// TIA Portal project "DrillingMachineS7300_S71500" (V15.1)

(* hardware
DEVICE "S7300/ET200M-Station_1"  S7-300 station
   slot 0: "Profilschiene_0"  Rail  6ES7 390-1***0-0AA0
   slot 2: "PLC_1"  CPU 315-2 PN/DP  6ES7 315-2EH14-0AB0  V3.2
      slot 2: "PROFINET-Schnittstelle_1"  PN-IO
         slot 1: "Port_1"  Port
         slot 2: "Port_2"  Port
   slot 4: "DI 32x24VDC_1"  DI32 x 24VDC  6ES7 321-1BL00-0AA0
   slot 5: "DO 32x24VDC/0.5A_1"  DO32 x 24VDC / 0.5A  6ES7 322-1BL00-0AA0
   slot 6: "AI 2x12BIT_1"  AI2 x 12 bits  6ES7 331-7KB02-0AB0
   slot 7: "AO 4x12BIT_1"  AO4 x 12 bits  6ES7 332-5HD01-0AB0
DEVICE "S71500/ET200MP-Station_1"  S7-1500 station
   slot 0: "Profilschiene_0"  Rack  6ES7 590-1***0-0AA0
   slot 1: "PLC_2"  CPU 1513-1 PN  6ES7 513-1AL02-0AB0  V2.6
      slot 3: "CPU-Display_1"  6ES7591-1AA00-0AA0
   slot 2: "DI 32x24VDC BA_1"  DI 32x24VDC BA  6ES7 521-1BL10-0AA0  V1.0
   slot 3: "DQ 32x24VDC/0.5A ST_1"  DQ 32x24VDC/0.5A ST  6ES7 522-1BL00-0AB0  V2.0
   slot 4: "AI 4xU/I/RTD/TC ST_1"  AI 4xU/I/RTD/TC ST  6ES7 531-7QD00-0AB0  V1.0
   slot 5: "AQ 4xU/I ST_1"  AQ 4xU/I ST  6ES7 532-5HD00-0AB0  V2.2
   slot 6: "DI 16x24VDC BA_1"  DI 16x24VDC BA  6ES7 521-1BH10-0AA0  V1.0
*)

// ===== PLC "PLC_1"  CPU 315-2 PN/DP =====

VAR_GLOBAL   // PLC tag table "Standard-Variablentabelle"
   "ControlOn" AT %M0.0 : Bool;
   "InitialPos" AT %M0.1 : Bool;
   "B14ClampingJaw1Min" AT %E2.6 : Bool;   // NC
   "B15ClampingJaw2Min" AT %E2.7 : Bool;   // NC
   "B16ClampingJaw3Min" AT %E3.0 : Bool;   // NC
   "B17ClampingJaw4Min" AT %E3.1 : Bool;   // NC
   "M13ClampingJawsToMax" AT %A2.5 : Bool;
END_VAR

VAR_GLOBAL   // PLC tag table "Variablentabelle aus XML_1"
   "S1ControlOn" AT %I0.0 : Bool;
   "S2ControlOff" AT %I0.1 : Bool;
   "S3Start" AT %I0.2 : Bool;
   "B1DrillMachVertMin" AT %I1.0 : Bool;   // NC
   "B2DrillMachVertMax" AT %I1.1 : Bool;   // NC
   "P1ControlOn" AT %Q0.0 : Bool;
   "M1DrillMachToMax" AT %Q1.0 : Bool;
   "M2DrillMachToMin" AT %Q1.1 : Bool;
   "M3DrillMachOn" AT %Q1.2 : Bool;
   "M4RotateDrillMachine" AT %Q1.3 : Bool;
   "RotationDrillMachStart" AT %Q1.4 : Bool;
   "B4DrillMachHorizMin" AT %I1.3 : Bool;   // NC
   "B3RotationDrillMachPos" AT %IW10 : Int;
   "RotationDrillMachNewPosReached" AT %I1.2 : Bool;
   "RotationDrillMachNewPos" AT %QW10 : Int;
   "B5DrillMachHorizMax" AT %I1.4 : Bool;   // NC
   "M5DrillMachHoriz" AT %Q1.5 : Bool;
   "DrillMachHorizStart" AT %Q1.6 : Bool;
   "B6FeedMinPos" AT %I1.5 : Bool;   // NC
   "B7FeedMaxPos" AT %I1.6 : Bool;   // NC
   "B8FeedDrillPos" AT %I1.7 : Bool;
   "M7FeedToMax" AT %Q1.7 : Bool;
   "M8FeedToMin" AT %Q2.0 : Bool;
   "M9GuideToMax" AT %Q2.1 : Bool;
   "M10GuideToMin" AT %Q2.2 : Bool;
   "B9GuideMinPos" AT %I2.0 : Bool;   // NC
   "B10GuideMaxPos" AT %I2.1 : Bool;   // NC
   "M11SliderToMax" AT %Q2.3 : Bool;
   "M12SliderToMin" AT %Q2.4 : Bool;
   "B11SliderMinPos" AT %I2.2 : Bool;   // NC
   "B12SliderMaxPos" AT %I2.3 : Bool;   // NC
   "B13MetalRodInSliderPos" AT %I2.4 : Bool;
   "B18DrillMachHorizPos" AT %IW12 : Word;
   "DrillMachHorizNewPos" AT %QW12 : Word;
   "DrillMachHorizNewPosReached" AT %I2.5 : Bool;
END_VAR

DATA_BLOCK "DrillMachineHorizPositioning_DB_FirstPos"   // DB1
{ S7_Optimized_Access := 'FALSE' }
VERSION : 0.1
// stored: InstanceOfName DrillMachineHorizPositioning
"DrillMachineHorizPositioning"
BEGIN
END_DATA_BLOCK

DATA_BLOCK "DrillMachineRotPositioning_DB_FirstPos"   // DB2
{ S7_Optimized_Access := 'FALSE' }
VERSION : 0.1
// stored: InstanceOfName DrillMachineRotationPositioning
"DrillMachineRotationPositioning"
BEGIN
END_DATA_BLOCK

DATA_BLOCK "DrillMachineHorizPositioning_DB_SecondPos"   // DB3
{ S7_Optimized_Access := 'FALSE' }
VERSION : 0.1
// stored: InstanceOfName DrillMachineHorizPositioning
"DrillMachineHorizPositioning"
BEGIN
END_DATA_BLOCK

DATA_BLOCK "DrillMachineRotPositioning_DB_SecondPos"   // DB4
{ S7_Optimized_Access := 'FALSE' }
VERSION : 0.1
// stored: InstanceOfName DrillMachineRotationPositioning
"DrillMachineRotationPositioning"
BEGIN
END_DATA_BLOCK

DATA_BLOCK "DrillMachineHorizPositioning_DB_ThirdPos"   // DB5
{ S7_Optimized_Access := 'FALSE' }
VERSION : 0.1
// stored: InstanceOfName DrillMachineHorizPositioning
"DrillMachineHorizPositioning"
BEGIN
END_DATA_BLOCK

DATA_BLOCK "DrillMachineRotPositioning_DB_ThirdPos"   // DB6
{ S7_Optimized_Access := 'FALSE' }
VERSION : 0.1
// stored: InstanceOfName DrillMachineRotationPositioning
"DrillMachineRotationPositioning"
BEGIN
END_DATA_BLOCK

DATA_BLOCK "StepsDB"   // DB7
{ S7_Optimized_Access := 'FALSE' }
VERSION : 0.1
// stored: InstanceOfName Steps
"Steps"
BEGIN
END_DATA_BLOCK

FUNCTION_BLOCK "Steps"   // FB1, FBD
{ S7_Optimized_Access := 'FALSE' }
VERSION : 0.1
   VAR
      NewPosHorizReachedHelper_0 : Bool;
      NewPosVertReachedHelper_0 : Bool;
      NewPosHorizReachedHelper_1 : Bool;
      NewPosVertReachedHelper_1 : Bool;
      NewPosHorizReachedHelper_2 : Bool;
      NewPosVertReachedHelper_2 : Bool;
      NewPosHorizReachedHelper_3 : Bool;
      NewPosVertReachedHelper_3 : Bool;
      Step1 : Bool;
      Step2 : Bool;
      Step3 : Bool;
      Step4 : Bool;
      Step5 : Bool;
      Step6 : Bool;
      Step7 : Bool;
      Step8 : Bool;
      Step9 : Bool;
      Step10 : Bool;
      Step11 : Bool;
      Step12 : Bool;
      Step12A : Bool;
      Step13 : Bool;
      Step14 : Bool;
      Step15 : Bool;
      Step15A : Bool;
      Step16 : Bool;
      Step17 : Bool;
      Step18 : Bool;
      Step19 : Bool;
      Step20 : Bool;
      InStepChain : Bool;
   END_VAR
   VAR_TEMP   // added for the SCL form of the ladder/FBD networks
      _w1 : Bool;
   END_VAR
BEGIN

REGION Network 1: Start
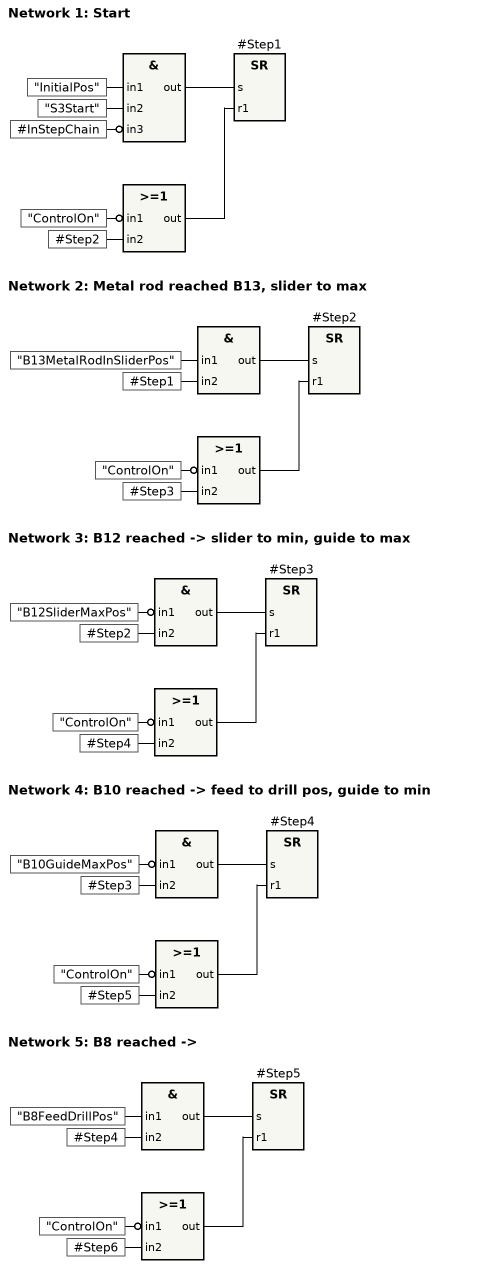
   IF "InitialPos" AND "S3Start" AND NOT #InStepChain THEN
       #Step1 := TRUE;   // SR flip-flop
   END_IF;
   IF NOT "ControlOn" OR #Step2 THEN #Step1 := FALSE; END_IF;
END_REGION

REGION Network 2: Metal rod reached B13, slider to max
   IF "B13MetalRodInSliderPos" AND #Step1 THEN
       #Step2 := TRUE;   // SR flip-flop
   END_IF;
   IF NOT "ControlOn" OR #Step3 THEN #Step2 := FALSE; END_IF;
END_REGION

REGION Network 3: B12 reached -> slider to min, guide to max
   // Slider stops with B11
   IF NOT "B12SliderMaxPos" AND #Step2 THEN
       #Step3 := TRUE;   // SR flip-flop
   END_IF;
   IF NOT "ControlOn" OR #Step4 THEN #Step3 := FALSE; END_IF;
END_REGION

REGION Network 4: B10 reached -> feed to drill pos, guide to min
   IF NOT "B10GuideMaxPos" AND #Step3 THEN
       #Step4 := TRUE;   // SR flip-flop
   END_IF;
   IF NOT "ControlOn" OR #Step5 THEN #Step4 := FALSE; END_IF;
END_REGION

REGION Network 5: B8 reached ->
   // guide stops with B9
   IF "B8FeedDrillPos" AND #Step4 THEN
       #Step5 := TRUE;   // SR flip-flop
   END_IF;
   IF NOT "ControlOn" OR #Step6 THEN #Step5 := FALSE; END_IF;
END_REGION

REGION Network 6: B9 also reached -> start drill cycle
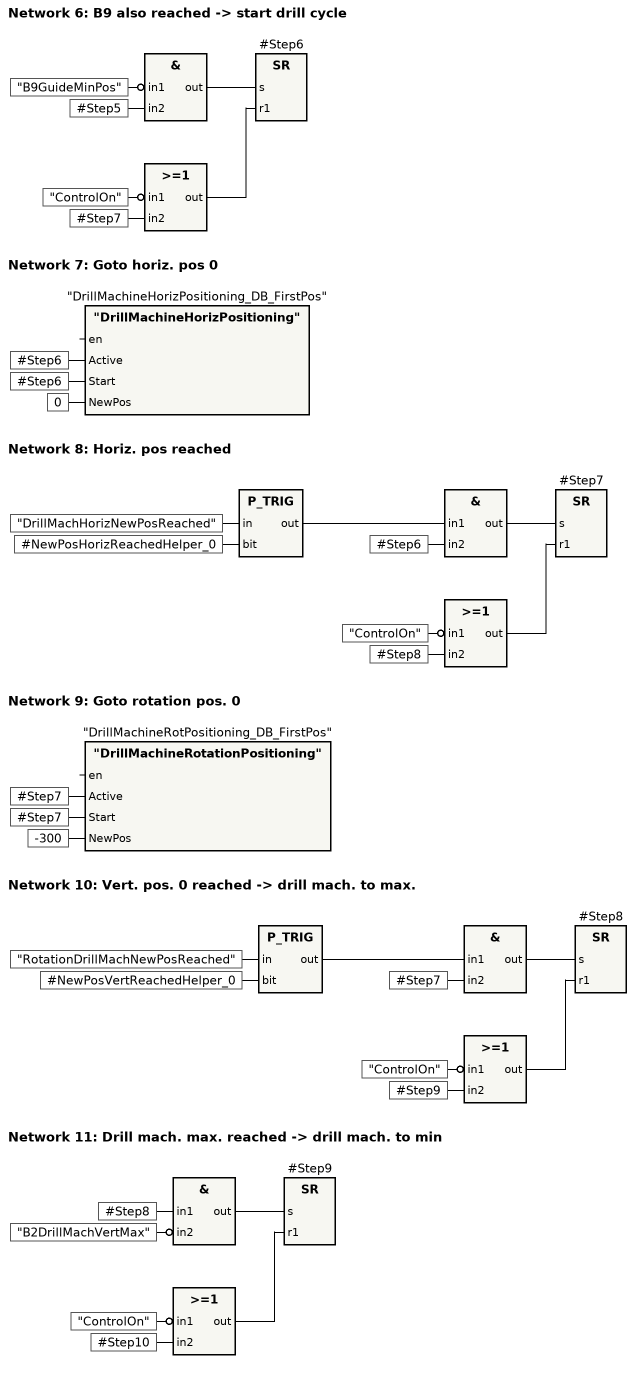
   IF NOT "B9GuideMinPos" AND #Step5 THEN
       #Step6 := TRUE;   // SR flip-flop
   END_IF;
   IF NOT "ControlOn" OR #Step7 THEN #Step6 := FALSE; END_IF;
END_REGION

REGION Network 7: Goto horiz. pos 0
   "DrillMachineHorizPositioning_DB_FirstPos"(Active := #Step6, Start := #Step6, NewPos := 0);   // "DrillMachineHorizPositioning"
END_REGION

REGION Network 8: Horiz. pos reached
   #_w1 := "DrillMachHorizNewPosReached" AND NOT #NewPosHorizReachedHelper_0;   // rising edge
   #NewPosHorizReachedHelper_0 := "DrillMachHorizNewPosReached";
   IF #_w1 AND #Step6 THEN
       #Step7 := TRUE;   // SR flip-flop
   END_IF;
   IF NOT "ControlOn" OR #Step8 THEN #Step7 := FALSE; END_IF;
END_REGION

REGION Network 9: Goto rotation pos. 0
   "DrillMachineRotPositioning_DB_FirstPos"(Active := #Step7, Start := #Step7, NewPos := -300);   // "DrillMachineRotationPositioning"
END_REGION

REGION Network 10: Vert. pos. 0 reached -> drill mach. to max.
   #_w1 := "RotationDrillMachNewPosReached" AND NOT #NewPosVertReachedHelper_0;   // rising edge
   #NewPosVertReachedHelper_0 := "RotationDrillMachNewPosReached";
   IF #_w1 AND #Step7 THEN
       #Step8 := TRUE;   // SR flip-flop
   END_IF;
   IF NOT "ControlOn" OR #Step9 THEN #Step8 := FALSE; END_IF;
END_REGION

REGION Network 11: Drill mach. max. reached -> drill mach. to min
   IF #Step8 AND NOT "B2DrillMachVertMax" THEN
       #Step9 := TRUE;   // SR flip-flop
   END_IF;
   IF NOT "ControlOn" OR #Step10 THEN #Step9 := FALSE; END_IF;
END_REGION

REGION Network 12: Min reached
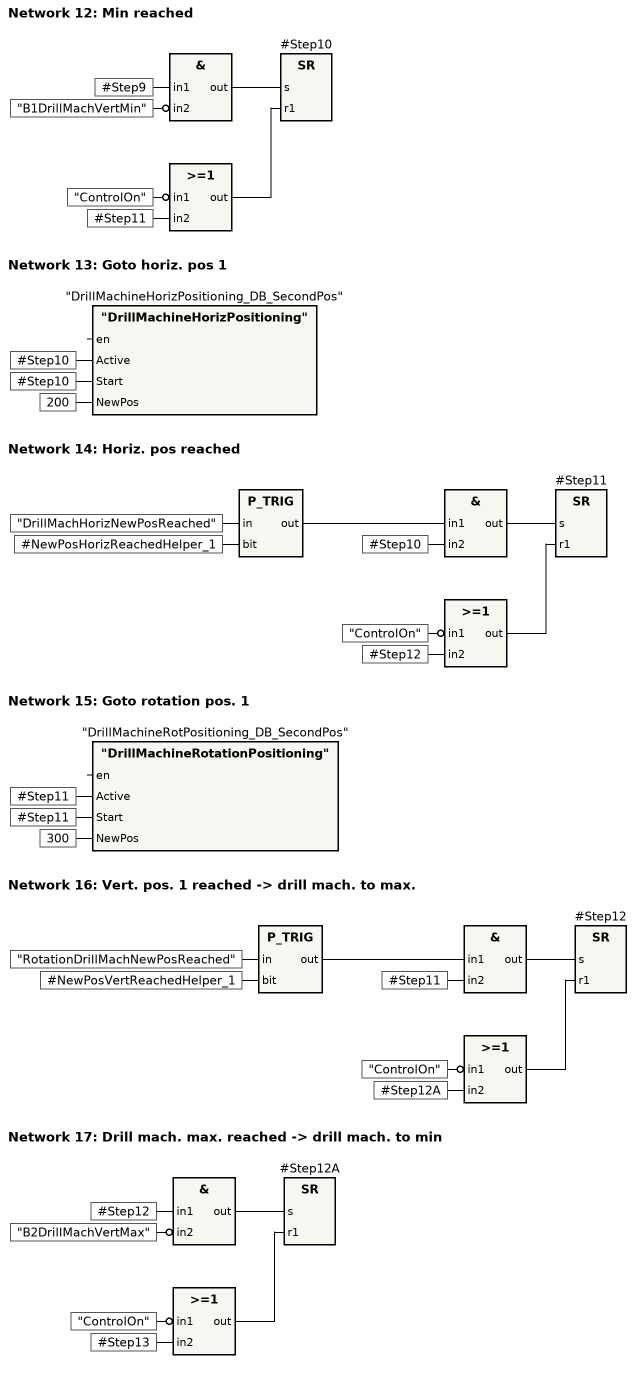
   IF #Step9 AND NOT "B1DrillMachVertMin" THEN
       #Step10 := TRUE;   // SR flip-flop
   END_IF;
   IF NOT "ControlOn" OR #Step11 THEN #Step10 := FALSE; END_IF;
END_REGION

REGION Network 13: Goto horiz. pos 1
   "DrillMachineHorizPositioning_DB_SecondPos"(Active := #Step10, Start := #Step10, NewPos := 200);   // "DrillMachineHorizPositioning"
END_REGION

REGION Network 14: Horiz. pos reached
   #_w1 := "DrillMachHorizNewPosReached" AND NOT #NewPosHorizReachedHelper_1;   // rising edge
   #NewPosHorizReachedHelper_1 := "DrillMachHorizNewPosReached";
   IF #_w1 AND #Step10 THEN
       #Step11 := TRUE;   // SR flip-flop
   END_IF;
   IF NOT "ControlOn" OR #Step12 THEN #Step11 := FALSE; END_IF;
END_REGION

REGION Network 15: Goto rotation pos. 1
   "DrillMachineRotPositioning_DB_SecondPos"(Active := #Step11, Start := #Step11, NewPos := 300);   // "DrillMachineRotationPositioning"
END_REGION

REGION Network 16: Vert. pos. 1 reached -> drill mach. to max.
   #_w1 := "RotationDrillMachNewPosReached" AND NOT #NewPosVertReachedHelper_1;   // rising edge
   #NewPosVertReachedHelper_1 := "RotationDrillMachNewPosReached";
   IF #_w1 AND #Step11 THEN
       #Step12 := TRUE;   // SR flip-flop
   END_IF;
   IF NOT "ControlOn" OR #Step12A THEN #Step12 := FALSE; END_IF;
END_REGION

REGION Network 17: Drill mach. max. reached -> drill mach. to min
   IF #Step12 AND NOT "B2DrillMachVertMax" THEN
       #Step12A := TRUE;   // SR flip-flop
   END_IF;
   IF NOT "ControlOn" OR #Step13 THEN #Step12A := FALSE; END_IF;
END_REGION

REGION Network 18: Min reached
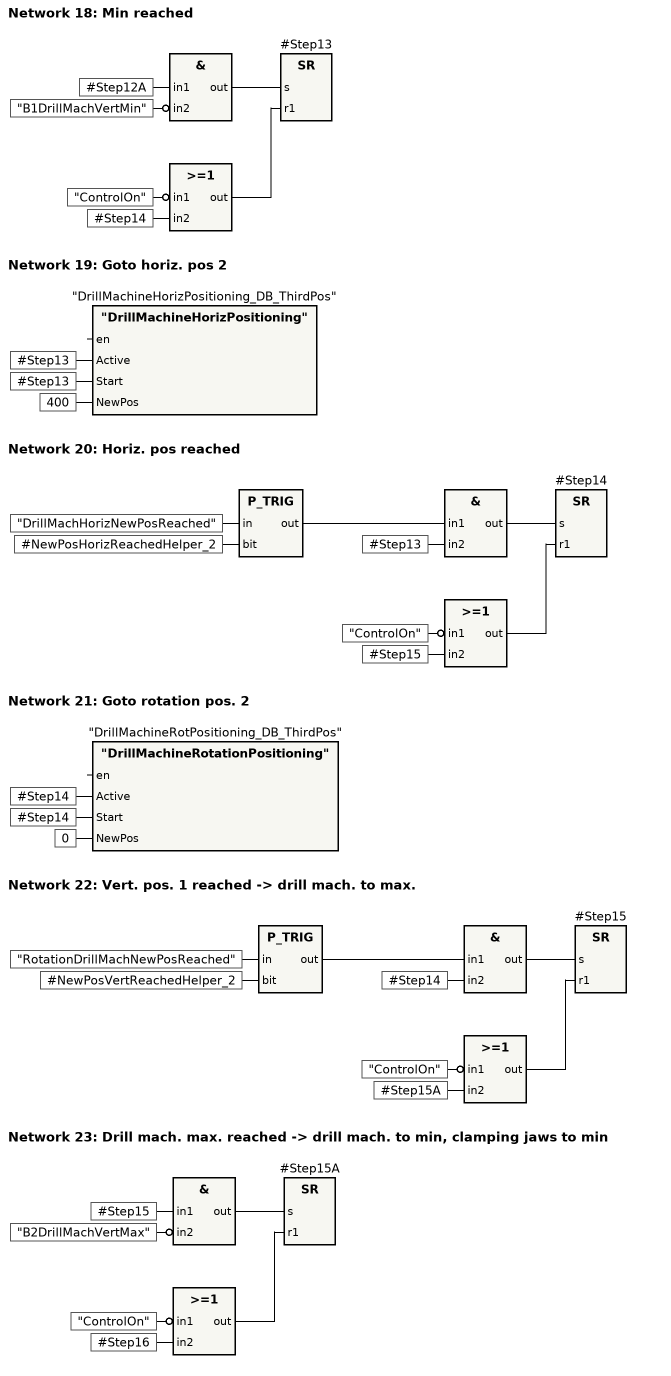
   IF #Step12A AND NOT "B1DrillMachVertMin" THEN
       #Step13 := TRUE;   // SR flip-flop
   END_IF;
   IF NOT "ControlOn" OR #Step14 THEN #Step13 := FALSE; END_IF;
END_REGION

REGION Network 19: Goto horiz. pos 2
   "DrillMachineHorizPositioning_DB_ThirdPos"(Active := #Step13, Start := #Step13, NewPos := 400);   // "DrillMachineHorizPositioning"
END_REGION

REGION Network 20: Horiz. pos reached
   #_w1 := "DrillMachHorizNewPosReached" AND NOT #NewPosHorizReachedHelper_2;   // rising edge
   #NewPosHorizReachedHelper_2 := "DrillMachHorizNewPosReached";
   IF #_w1 AND #Step13 THEN
       #Step14 := TRUE;   // SR flip-flop
   END_IF;
   IF NOT "ControlOn" OR #Step15 THEN #Step14 := FALSE; END_IF;
END_REGION

REGION Network 21: Goto rotation pos. 2
   "DrillMachineRotPositioning_DB_ThirdPos"(Active := #Step14, Start := #Step14, NewPos := 0);   // "DrillMachineRotationPositioning"
END_REGION

REGION Network 22: Vert. pos. 1 reached -> drill mach. to max.
   #_w1 := "RotationDrillMachNewPosReached" AND NOT #NewPosVertReachedHelper_2;   // rising edge
   #NewPosVertReachedHelper_2 := "RotationDrillMachNewPosReached";
   IF #_w1 AND #Step14 THEN
       #Step15 := TRUE;   // SR flip-flop
   END_IF;
   IF NOT "ControlOn" OR #Step15A THEN #Step15 := FALSE; END_IF;
END_REGION

REGION Network 23: Drill mach. max. reached -> drill mach. to min, clamping jaws to min
   IF #Step15 AND NOT "B2DrillMachVertMax" THEN
       #Step15A := TRUE;   // SR flip-flop
   END_IF;
   IF NOT "ControlOn" OR #Step16 THEN #Step15A := FALSE; END_IF;
END_REGION

REGION Network 24: Min reached -> Feed to max.
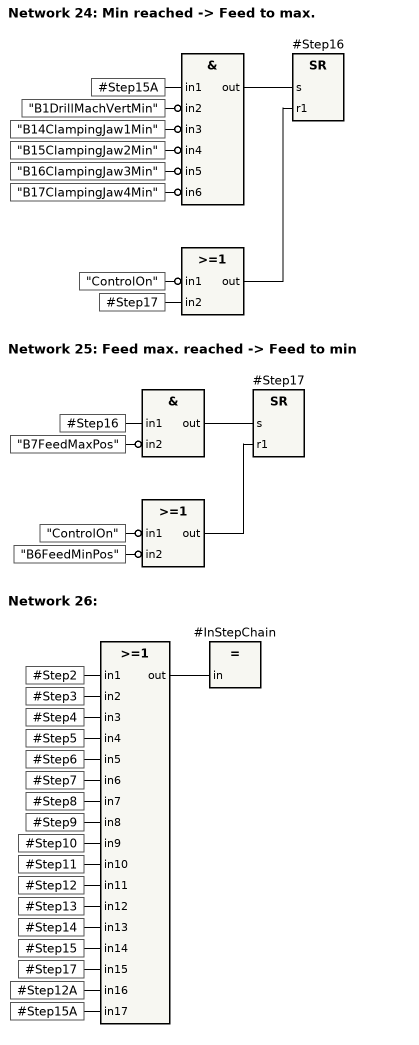
   IF #Step15A AND NOT "B1DrillMachVertMin" AND NOT "B14ClampingJaw1Min" AND NOT "B15ClampingJaw2Min" AND NOT "B16ClampingJaw3Min" AND NOT "B17ClampingJaw4Min" THEN
       #Step16 := TRUE;   // SR flip-flop
   END_IF;
   IF NOT "ControlOn" OR #Step17 THEN #Step16 := FALSE; END_IF;
END_REGION

REGION Network 25: Feed max. reached -> Feed to min
   IF #Step16 AND NOT "B7FeedMaxPos" THEN
       #Step17 := TRUE;   // SR flip-flop
   END_IF;
   IF NOT "ControlOn" OR NOT "B6FeedMinPos" THEN #Step17 := FALSE; END_IF;
END_REGION

REGION Network 26
   #InStepChain := #Step2 OR #Step3 OR #Step4 OR #Step5 OR #Step6 OR #Step7 OR #Step8 OR #Step9 OR #Step10 OR #Step11 OR #Step12 OR #Step13 OR #Step14 OR #Step15 OR #Step17 OR #Step12A OR #Step15A;
END_REGION
END_FUNCTION_BLOCK

FUNCTION_BLOCK "DrillMachineHorizPositioning"   // FB2, FBD
{ S7_Optimized_Access := 'FALSE' }
VERSION : 0.1
   VAR_INPUT
      Active : Bool;
      Start : Bool;
      NewPos : Int := 0;
   END_VAR
   VAR
      PosEdgeStartHelper : Bool;
      PosEdgeStart : Bool;
   END_VAR
   VAR_TEMP   // added for the SCL form of the ladder/FBD networks
      _w1 : Bool;
   END_VAR
BEGIN

REGION Network 1: Active?
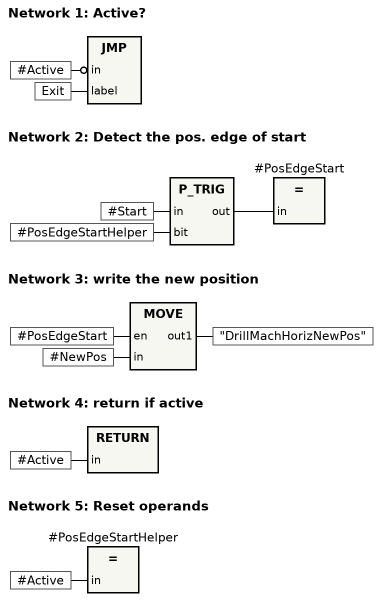
   IF NOT #Active THEN GOTO Exit; END_IF;
END_REGION

REGION Network 2: Detect the pos. edge of start
   #_w1 := #Start AND NOT #PosEdgeStartHelper;   // rising edge
   #PosEdgeStartHelper := #Start;
   #PosEdgeStart := #_w1;
END_REGION

REGION Network 3: write the new position
   IF #PosEdgeStart THEN "DrillMachHorizNewPos" := #NewPos; END_IF;
END_REGION

REGION Network 4: return if active
   IF #Active THEN
       ENO := TRUE;
       RETURN;
   END_IF;
END_REGION

REGION Network 5: Reset operands
   Exit:
   #PosEdgeStartHelper := #Active;
END_REGION
END_FUNCTION_BLOCK

FUNCTION_BLOCK "DrillMachineRotationPositioning"   // FB3, FBD
{ S7_Optimized_Access := 'FALSE' }
VERSION : 0.1
   VAR_INPUT
      Active : Bool;
      Start : Bool;
      NewPos : Int := 0;
   END_VAR
   VAR
      PosEdgeStartHelper : Bool;
      PosEdgeStart : Bool;
   END_VAR
   VAR_TEMP   // added for the SCL form of the ladder/FBD networks
      _w1 : Bool;
   END_VAR
BEGIN

REGION Network 1
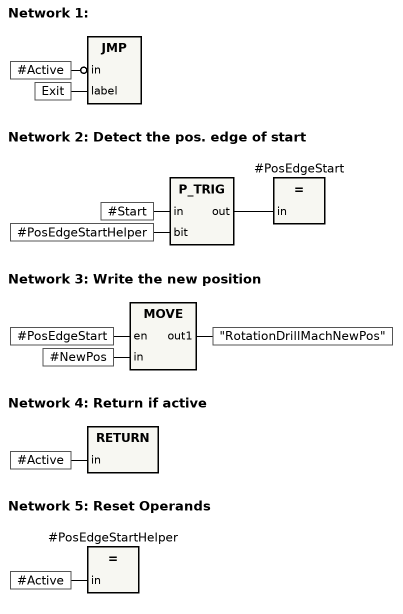
   IF NOT #Active THEN GOTO Exit; END_IF;
END_REGION

REGION Network 2: Detect the pos. edge of start
   #_w1 := #Start AND NOT #PosEdgeStartHelper;   // rising edge
   #PosEdgeStartHelper := #Start;
   #PosEdgeStart := #_w1;
END_REGION

REGION Network 3: Write the new position
   IF #PosEdgeStart THEN "RotationDrillMachNewPos" := #NewPos; END_IF;
END_REGION

REGION Network 4: Return if active
   IF #Active THEN
       ENO := TRUE;
       RETURN;
   END_IF;
END_REGION

REGION Network 5: Reset Operands
   Exit:
   #PosEdgeStartHelper := #Active;
END_REGION
END_FUNCTION_BLOCK

FUNCTION "Settings" : Void   // FC1, FBD
{ S7_Optimized_Access := 'FALSE' }
VERSION : 0.1
BEGIN

REGION Network 1: Slider to max
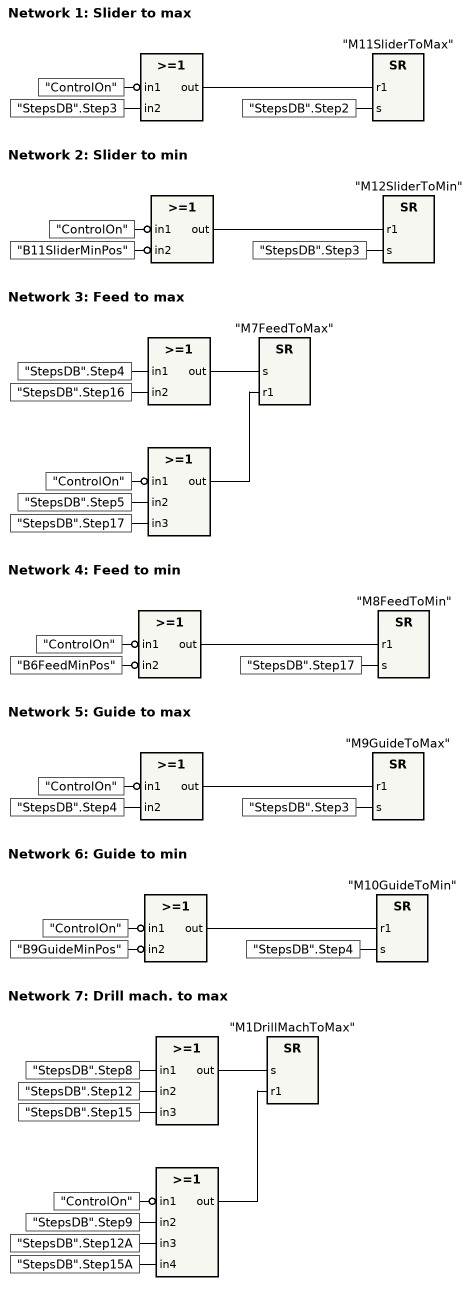
   IF "StepsDB".Step2 THEN
       "M11SliderToMax" := TRUE;   // SR flip-flop
   END_IF;
   IF NOT "ControlOn" OR "StepsDB".Step3 THEN "M11SliderToMax" := FALSE; END_IF;
END_REGION

REGION Network 2: Slider to min
   IF "StepsDB".Step3 THEN
       "M12SliderToMin" := TRUE;   // SR flip-flop
   END_IF;
   IF NOT "ControlOn" OR NOT "B11SliderMinPos" THEN "M12SliderToMin" := FALSE; END_IF;
END_REGION

REGION Network 3: Feed to max
   IF "StepsDB".Step4 OR "StepsDB".Step16 THEN
       "M7FeedToMax" := TRUE;   // SR flip-flop
   END_IF;
   IF NOT "ControlOn" OR "StepsDB".Step5 OR "StepsDB".Step17 THEN "M7FeedToMax" := FALSE; END_IF;
END_REGION

REGION Network 4: Feed to min
   IF "StepsDB".Step17 THEN
       "M8FeedToMin" := TRUE;   // SR flip-flop
   END_IF;
   IF NOT "ControlOn" OR NOT "B6FeedMinPos" THEN "M8FeedToMin" := FALSE; END_IF;
END_REGION

REGION Network 5: Guide to max
   IF "StepsDB".Step3 THEN
       "M9GuideToMax" := TRUE;   // SR flip-flop
   END_IF;
   IF NOT "ControlOn" OR "StepsDB".Step4 THEN "M9GuideToMax" := FALSE; END_IF;
END_REGION

REGION Network 6: Guide to min
   IF "StepsDB".Step4 THEN
       "M10GuideToMin" := TRUE;   // SR flip-flop
   END_IF;
   IF NOT "ControlOn" OR NOT "B9GuideMinPos" THEN "M10GuideToMin" := FALSE; END_IF;
END_REGION

REGION Network 7: Drill mach. to max
   IF "StepsDB".Step8 OR "StepsDB".Step12 OR "StepsDB".Step15 THEN
       "M1DrillMachToMax" := TRUE;   // SR flip-flop
   END_IF;
   IF NOT "ControlOn" OR "StepsDB".Step9 OR "StepsDB".Step12A OR "StepsDB".Step15A THEN
       "M1DrillMachToMax" := FALSE;
   END_IF;
END_REGION

REGION Network 8: Drill mach. to min
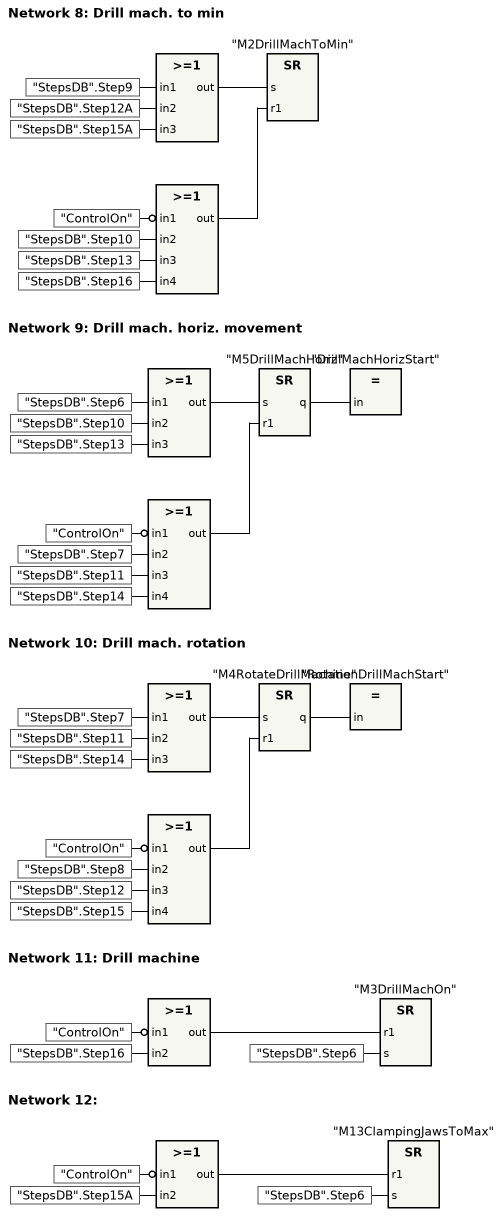
   IF "StepsDB".Step9 OR "StepsDB".Step12A OR "StepsDB".Step15A THEN
       "M2DrillMachToMin" := TRUE;   // SR flip-flop
   END_IF;
   IF NOT "ControlOn" OR "StepsDB".Step10 OR "StepsDB".Step13 OR "StepsDB".Step16 THEN
       "M2DrillMachToMin" := FALSE;
   END_IF;
END_REGION

REGION Network 9: Drill mach. horiz. movement
   IF "StepsDB".Step6 OR "StepsDB".Step10 OR "StepsDB".Step13 THEN
       "M5DrillMachHoriz" := TRUE;   // SR flip-flop
   END_IF;
   IF NOT "ControlOn" OR "StepsDB".Step7 OR "StepsDB".Step11 OR "StepsDB".Step14 THEN
       "M5DrillMachHoriz" := FALSE;
   END_IF;
   "DrillMachHorizStart" := "M5DrillMachHoriz";
END_REGION

REGION Network 10: Drill mach. rotation
   IF "StepsDB".Step7 OR "StepsDB".Step11 OR "StepsDB".Step14 THEN
       "M4RotateDrillMachine" := TRUE;   // SR flip-flop
   END_IF;
   IF NOT "ControlOn" OR "StepsDB".Step8 OR "StepsDB".Step12 OR "StepsDB".Step15 THEN
       "M4RotateDrillMachine" := FALSE;
   END_IF;
   "RotationDrillMachStart" := "M4RotateDrillMachine";
END_REGION

REGION Network 11: Drill machine
   IF "StepsDB".Step6 THEN
       "M3DrillMachOn" := TRUE;   // SR flip-flop
   END_IF;
   IF NOT "ControlOn" OR "StepsDB".Step16 THEN "M3DrillMachOn" := FALSE; END_IF;
END_REGION

REGION Network 12
   IF "StepsDB".Step6 THEN
       "M13ClampingJawsToMax" := TRUE;   // SR flip-flop
   END_IF;
   IF NOT "ControlOn" OR "StepsDB".Step15A THEN "M13ClampingJawsToMax" := FALSE; END_IF;
END_REGION
END_FUNCTION

ORGANIZATION_BLOCK "Main"   // OB1, FBD
TITLE = "Main Program Sweep (Cycle)"
{ S7_Optimized_Access := 'FALSE' }
VERSION : 0.1
   VAR_TEMP
      OB1_EV_CLASS : Byte;   // Bits 0-3 = 1 (Coming event), Bits 4-7 = 1 (Event class 1)
      OB1_SCAN_1 : Byte;   // 1 (Cold restart scan 1 of OB 1), 3 (Scan 2-n of OB 1)
      OB1_PRIORITY : Byte;   // Priority of OB Execution
      OB1_OB_NUMBR : Byte;   // 1 (Organization block 1, OB1)
      OB1_RESERVED_1 : Byte;   // Reserved for system
      OB1_RESERVED_2 : Byte;   // Reserved for system
      OB1_PREV_CYCLE : Int;   // Cycle time of previous OB1 scan (milliseconds)
      OB1_MIN_CYCLE : Int;   // Minimum cycle time of OB1 (milliseconds)
      OB1_MAX_CYCLE : Int;   // Maximum cycle time of OB1 (milliseconds)
      OB1_DATE_TIME : Date_And_Time;   // Date and time OB1 started
   END_VAR
BEGIN

REGION Network 1
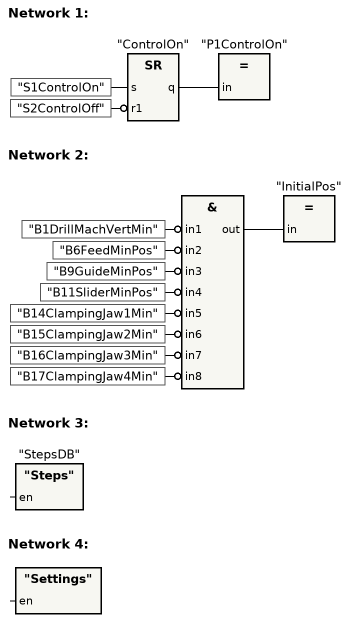
   IF "S1ControlOn" THEN
       "ControlOn" := TRUE;   // SR flip-flop
   END_IF;
   IF NOT "S2ControlOff" THEN "ControlOn" := FALSE; END_IF;
   "P1ControlOn" := "ControlOn";
END_REGION

REGION Network 2
   "InitialPos" := NOT "B1DrillMachVertMin" AND NOT "B6FeedMinPos" AND NOT "B9GuideMinPos" AND NOT "B11SliderMinPos" AND NOT "B14ClampingJaw1Min" AND NOT "B15ClampingJaw2Min" AND NOT "B16ClampingJaw3Min" AND NOT "B17ClampingJaw4Min";
END_REGION

REGION Network 3
   "StepsDB"();   // "Steps"
END_REGION

REGION Network 4
   "Settings"();
END_REGION
END_ORGANIZATION_BLOCK

// ===== PLC "PLC_2"  CPU 1513-1 PN =====

VAR_GLOBAL   // PLC tag table "Standard-Variablentabelle"
   "S1ControlOn" AT %I0.0 : Bool;
   "S2ControlOff" AT %I0.1 : Bool;
   "S3Start" AT %I0.2 : Bool;
   "B1DrillMachVertMin" AT %I1.0 : Bool;   // NC
   "B2DrillMachVertMax" AT %I1.1 : Bool;   // NC
   "P1ControlOn" AT %Q0.0 : Bool;
   "M1DrillMachToMax" AT %Q1.0 : Bool;
   "M2DrillMachToMin" AT %Q1.1 : Bool;
   "M3DrillMachOn" AT %Q1.2 : Bool;
   "M4RotateDrillMachine" AT %Q1.3 : Bool;
   "RotationDrillMachStart" AT %Q1.4 : Bool;
   "B4DrillMachHorizMin" AT %I1.3 : Bool;   // NC
   "B3RotationDrillMachPos" AT %IW10 : Int;
   "RotationDrillMachNewPosReached" AT %I1.2 : Bool;
   "RotationDrillMachNewPos" AT %QW10 : Int;
   "B5DrillMachHorizMax" AT %I1.4 : Bool;   // NC
   "M5DrillMachHoriz" AT %Q1.5 : Bool;
   "DrillMachHorizStart" AT %Q1.6 : Bool;
   "B6FeedMinPos" AT %I1.5 : Bool;   // NC
   "B7FeedMaxPos" AT %I1.6 : Bool;   // NC
   "B8FeedDrillPos" AT %I1.7 : Bool;
   "M7FeedToMax" AT %Q1.7 : Bool;
   "M8FeedToMin" AT %Q2.0 : Bool;
   "M9GuideToMax" AT %Q2.1 : Bool;
   "M10GuideToMin" AT %Q2.2 : Bool;
   "B9GuideMinPos" AT %I2.0 : Bool;   // NC
   "B10GuideMaxPos" AT %I2.1 : Bool;   // NC
   "M11SliderToMax" AT %Q2.3 : Bool;
   "M12SliderToMin" AT %Q2.4 : Bool;
   "B11SliderMinPos" AT %I2.2 : Bool;   // NC
   "B12SliderMaxPos" AT %I2.3 : Bool;   // NC
   "B13MetalRodInSliderPos" AT %I2.4 : Bool;
   "B18DrillMachHorizPos" AT %IW12 : Word;
   "DrillMachHorizNewPos" AT %QW12 : Word;
   "DrillMachHorizNewPosReached" AT %I2.5 : Bool;
   "ControlOn" AT %M0.0 : Bool;
   "InitialPos" AT %M0.1 : Bool;
   "B14ClampingJaw1Min" AT %E2.6 : Bool;   // NC
   "B15ClampingJaw2Min" AT %E2.7 : Bool;   // NC
   "B16ClampingJaw3Min" AT %E3.0 : Bool;   // NC
   "B17ClampingJaw4Min" AT %E3.1 : Bool;   // NC
   "M13ClampingJawsToMax" AT %A2.5 : Bool;
END_VAR

DATA_BLOCK "DrillMachineHorizPositioning_DB_FirstPos"   // DB1
{ S7_Optimized_Access := 'FALSE' }
VERSION : 0.1
// stored: InstanceOfName DrillMachineHorizPositioning
"DrillMachineHorizPositioning"
BEGIN
END_DATA_BLOCK

DATA_BLOCK "DrillMachineRotPositioning_DB_FirstPos"   // DB2
{ S7_Optimized_Access := 'FALSE' }
VERSION : 0.1
// stored: InstanceOfName DrillMachineRotationPositioning
"DrillMachineRotationPositioning"
BEGIN
END_DATA_BLOCK

DATA_BLOCK "DrillMachineHorizPositioning_DB_SecondPos"   // DB3
{ S7_Optimized_Access := 'FALSE' }
VERSION : 0.1
// stored: InstanceOfName DrillMachineHorizPositioning
"DrillMachineHorizPositioning"
BEGIN
END_DATA_BLOCK

DATA_BLOCK "DrillMachineRotPositioning_DB_SecondPos"   // DB4
{ S7_Optimized_Access := 'FALSE' }
VERSION : 0.1
// stored: InstanceOfName DrillMachineRotationPositioning
"DrillMachineRotationPositioning"
BEGIN
END_DATA_BLOCK

DATA_BLOCK "DrillMachineHorizPositioning_DB_ThirdPos"   // DB5
{ S7_Optimized_Access := 'FALSE' }
VERSION : 0.1
// stored: InstanceOfName DrillMachineHorizPositioning
"DrillMachineHorizPositioning"
BEGIN
END_DATA_BLOCK

DATA_BLOCK "DrillMachineRotPositioning_DB_ThirdPos"   // DB6
{ S7_Optimized_Access := 'FALSE' }
VERSION : 0.1
// stored: InstanceOfName DrillMachineRotationPositioning
"DrillMachineRotationPositioning"
BEGIN
END_DATA_BLOCK

DATA_BLOCK "StepsDB"   // DB7
{ S7_Optimized_Access := 'FALSE' }
VERSION : 0.1
// stored: InstanceOfName Steps
"Steps"
BEGIN
END_DATA_BLOCK

FUNCTION_BLOCK "Steps"   // FB1, FBD
{ S7_Optimized_Access := 'FALSE' }
VERSION : 0.1
   VAR
      NewPosHorizReachedHelper_0 : Bool;
      NewPosVertReachedHelper_0 : Bool;
      NewPosHorizReachedHelper_1 : Bool;
      NewPosVertReachedHelper_1 : Bool;
      NewPosHorizReachedHelper_2 : Bool;
      NewPosVertReachedHelper_2 : Bool;
      NewPosHorizReachedHelper_3 : Bool;
      NewPosVertReachedHelper_3 : Bool;
      Step1 : Bool;
      Step2 : Bool;
      Step3 : Bool;
      Step4 : Bool;
      Step5 : Bool;
      Step6 : Bool;
      Step7 : Bool;
      Step8 : Bool;
      Step9 : Bool;
      Step10 : Bool;
      Step11 : Bool;
      Step12 : Bool;
      Step12A : Bool;
      Step13 : Bool;
      Step14 : Bool;
      Step15 : Bool;
      Step15A : Bool;
      Step16 : Bool;
      Step17 : Bool;
      Step18 : Bool;
      Step19 : Bool;
      Step20 : Bool;
      InStepChain : Bool;
   END_VAR
   VAR_TEMP   // added for the SCL form of the ladder/FBD networks
      _w1 : Bool;
   END_VAR
BEGIN

REGION Network 1: Start
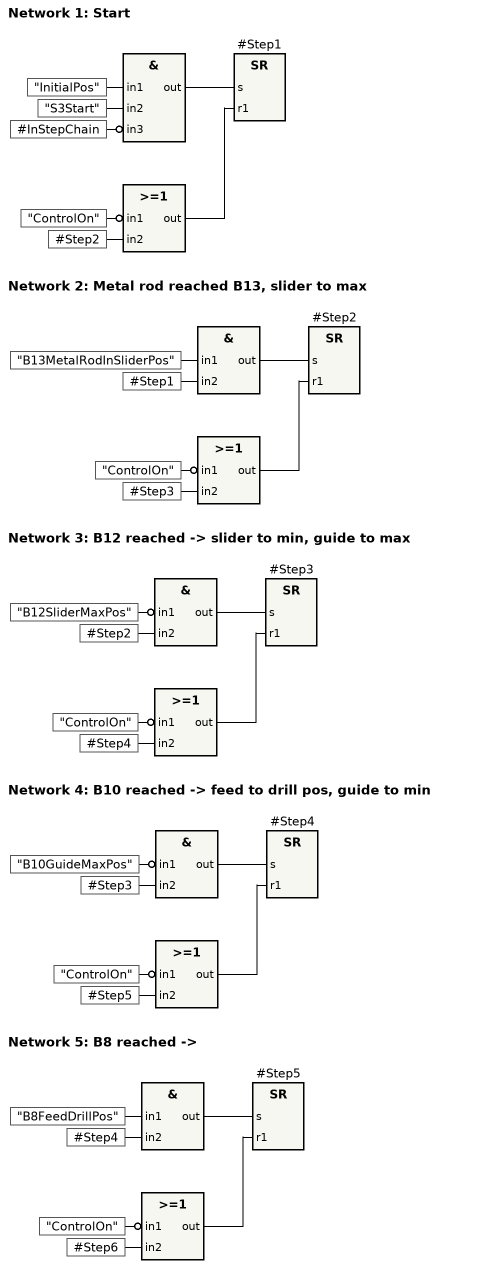
   IF "InitialPos" AND "S3Start" AND NOT #InStepChain THEN
       #Step1 := TRUE;   // SR flip-flop
   END_IF;
   IF NOT "ControlOn" OR #Step2 THEN #Step1 := FALSE; END_IF;
END_REGION

REGION Network 2: Metal rod reached B13, slider to max
   IF "B13MetalRodInSliderPos" AND #Step1 THEN
       #Step2 := TRUE;   // SR flip-flop
   END_IF;
   IF NOT "ControlOn" OR #Step3 THEN #Step2 := FALSE; END_IF;
END_REGION

REGION Network 3: B12 reached -> slider to min, guide to max
   // Slider stops with B11
   IF NOT "B12SliderMaxPos" AND #Step2 THEN
       #Step3 := TRUE;   // SR flip-flop
   END_IF;
   IF NOT "ControlOn" OR #Step4 THEN #Step3 := FALSE; END_IF;
END_REGION

REGION Network 4: B10 reached -> feed to drill pos, guide to min
   IF NOT "B10GuideMaxPos" AND #Step3 THEN
       #Step4 := TRUE;   // SR flip-flop
   END_IF;
   IF NOT "ControlOn" OR #Step5 THEN #Step4 := FALSE; END_IF;
END_REGION

REGION Network 5: B8 reached ->
   // guide stops with B9
   IF "B8FeedDrillPos" AND #Step4 THEN
       #Step5 := TRUE;   // SR flip-flop
   END_IF;
   IF NOT "ControlOn" OR #Step6 THEN #Step5 := FALSE; END_IF;
END_REGION

REGION Network 6: B9 also reached -> start drill cycle
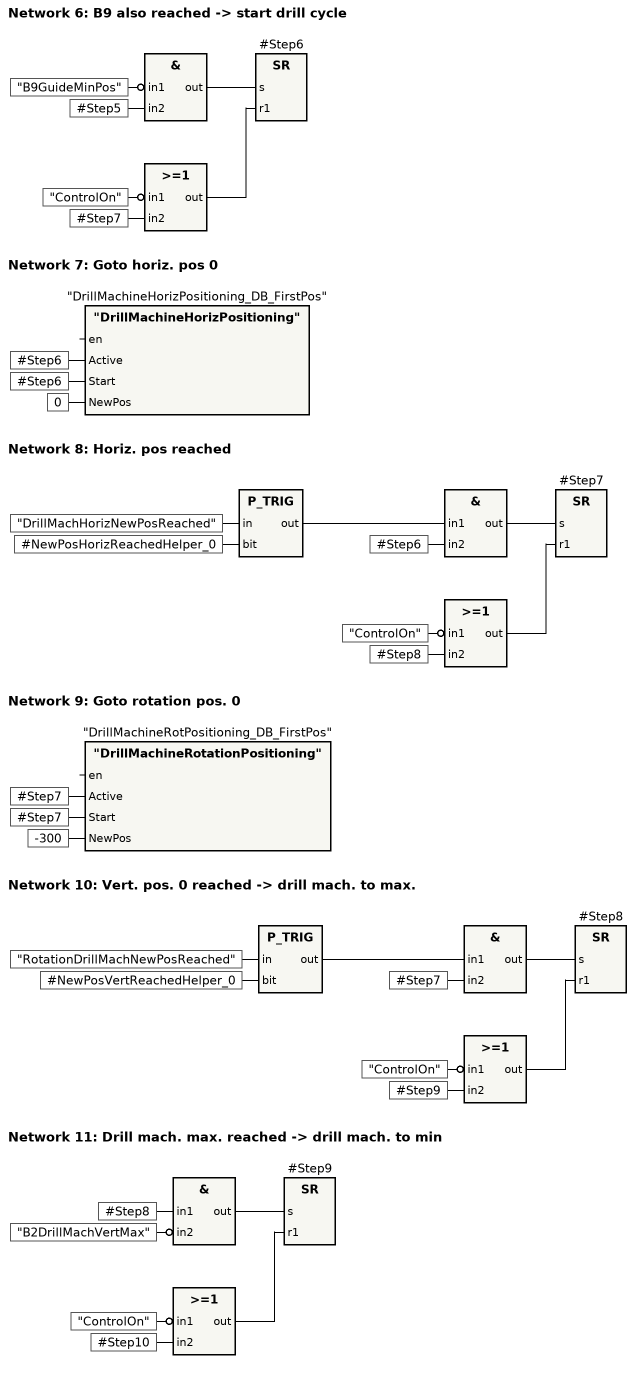
   IF NOT "B9GuideMinPos" AND #Step5 THEN
       #Step6 := TRUE;   // SR flip-flop
   END_IF;
   IF NOT "ControlOn" OR #Step7 THEN #Step6 := FALSE; END_IF;
END_REGION

REGION Network 7: Goto horiz. pos 0
   "DrillMachineHorizPositioning_DB_FirstPos"(Active := #Step6, Start := #Step6, NewPos := 0);   // "DrillMachineHorizPositioning"
END_REGION

REGION Network 8: Horiz. pos reached
   #_w1 := "DrillMachHorizNewPosReached" AND NOT #NewPosHorizReachedHelper_0;   // rising edge
   #NewPosHorizReachedHelper_0 := "DrillMachHorizNewPosReached";
   IF #_w1 AND #Step6 THEN
       #Step7 := TRUE;   // SR flip-flop
   END_IF;
   IF NOT "ControlOn" OR #Step8 THEN #Step7 := FALSE; END_IF;
END_REGION

REGION Network 9: Goto rotation pos. 0
   "DrillMachineRotPositioning_DB_FirstPos"(Active := #Step7, Start := #Step7, NewPos := -300);   // "DrillMachineRotationPositioning"
END_REGION

REGION Network 10: Vert. pos. 0 reached -> drill mach. to max.
   #_w1 := "RotationDrillMachNewPosReached" AND NOT #NewPosVertReachedHelper_0;   // rising edge
   #NewPosVertReachedHelper_0 := "RotationDrillMachNewPosReached";
   IF #_w1 AND #Step7 THEN
       #Step8 := TRUE;   // SR flip-flop
   END_IF;
   IF NOT "ControlOn" OR #Step9 THEN #Step8 := FALSE; END_IF;
END_REGION

REGION Network 11: Drill mach. max. reached -> drill mach. to min
   IF #Step8 AND NOT "B2DrillMachVertMax" THEN
       #Step9 := TRUE;   // SR flip-flop
   END_IF;
   IF NOT "ControlOn" OR #Step10 THEN #Step9 := FALSE; END_IF;
END_REGION

REGION Network 12: Min reached
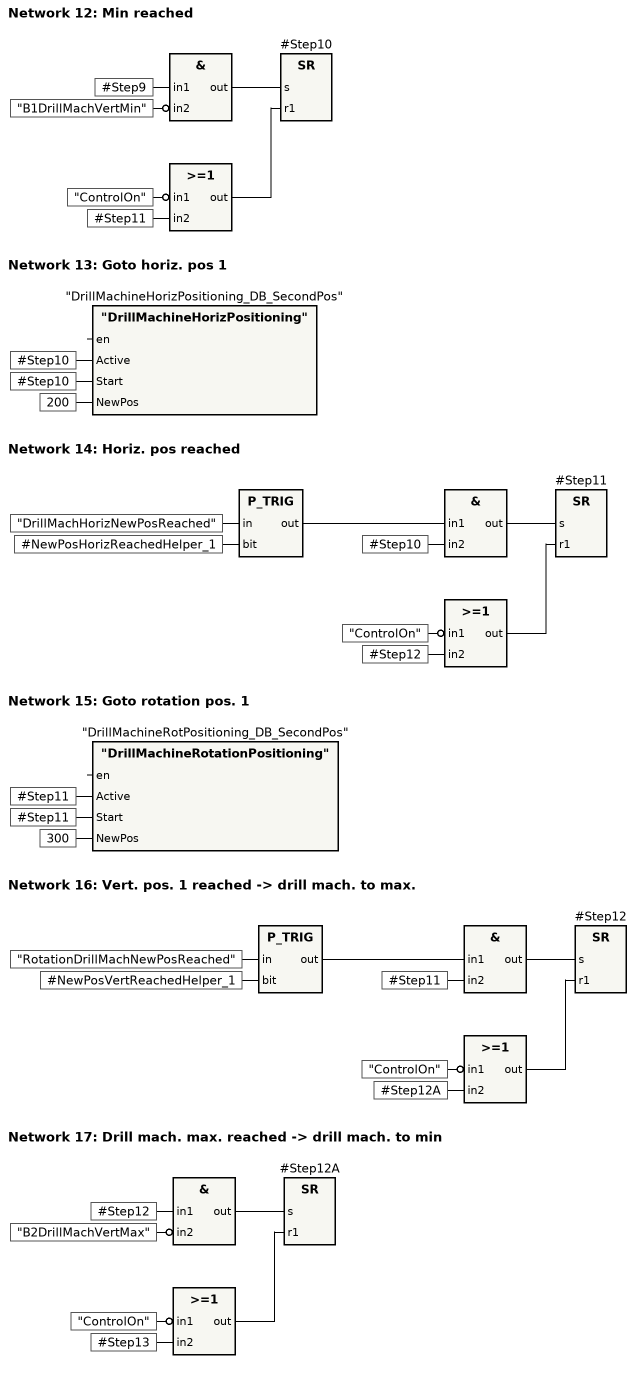
   IF #Step9 AND NOT "B1DrillMachVertMin" THEN
       #Step10 := TRUE;   // SR flip-flop
   END_IF;
   IF NOT "ControlOn" OR #Step11 THEN #Step10 := FALSE; END_IF;
END_REGION

REGION Network 13: Goto horiz. pos 1
   "DrillMachineHorizPositioning_DB_SecondPos"(Active := #Step10, Start := #Step10, NewPos := 200);   // "DrillMachineHorizPositioning"
END_REGION

REGION Network 14: Horiz. pos reached
   #_w1 := "DrillMachHorizNewPosReached" AND NOT #NewPosHorizReachedHelper_1;   // rising edge
   #NewPosHorizReachedHelper_1 := "DrillMachHorizNewPosReached";
   IF #_w1 AND #Step10 THEN
       #Step11 := TRUE;   // SR flip-flop
   END_IF;
   IF NOT "ControlOn" OR #Step12 THEN #Step11 := FALSE; END_IF;
END_REGION

REGION Network 15: Goto rotation pos. 1
   "DrillMachineRotPositioning_DB_SecondPos"(Active := #Step11, Start := #Step11, NewPos := 300);   // "DrillMachineRotationPositioning"
END_REGION

REGION Network 16: Vert. pos. 1 reached -> drill mach. to max.
   #_w1 := "RotationDrillMachNewPosReached" AND NOT #NewPosVertReachedHelper_1;   // rising edge
   #NewPosVertReachedHelper_1 := "RotationDrillMachNewPosReached";
   IF #_w1 AND #Step11 THEN
       #Step12 := TRUE;   // SR flip-flop
   END_IF;
   IF NOT "ControlOn" OR #Step12A THEN #Step12 := FALSE; END_IF;
END_REGION

REGION Network 17: Drill mach. max. reached -> drill mach. to min
   IF #Step12 AND NOT "B2DrillMachVertMax" THEN
       #Step12A := TRUE;   // SR flip-flop
   END_IF;
   IF NOT "ControlOn" OR #Step13 THEN #Step12A := FALSE; END_IF;
END_REGION

REGION Network 18: Min reached
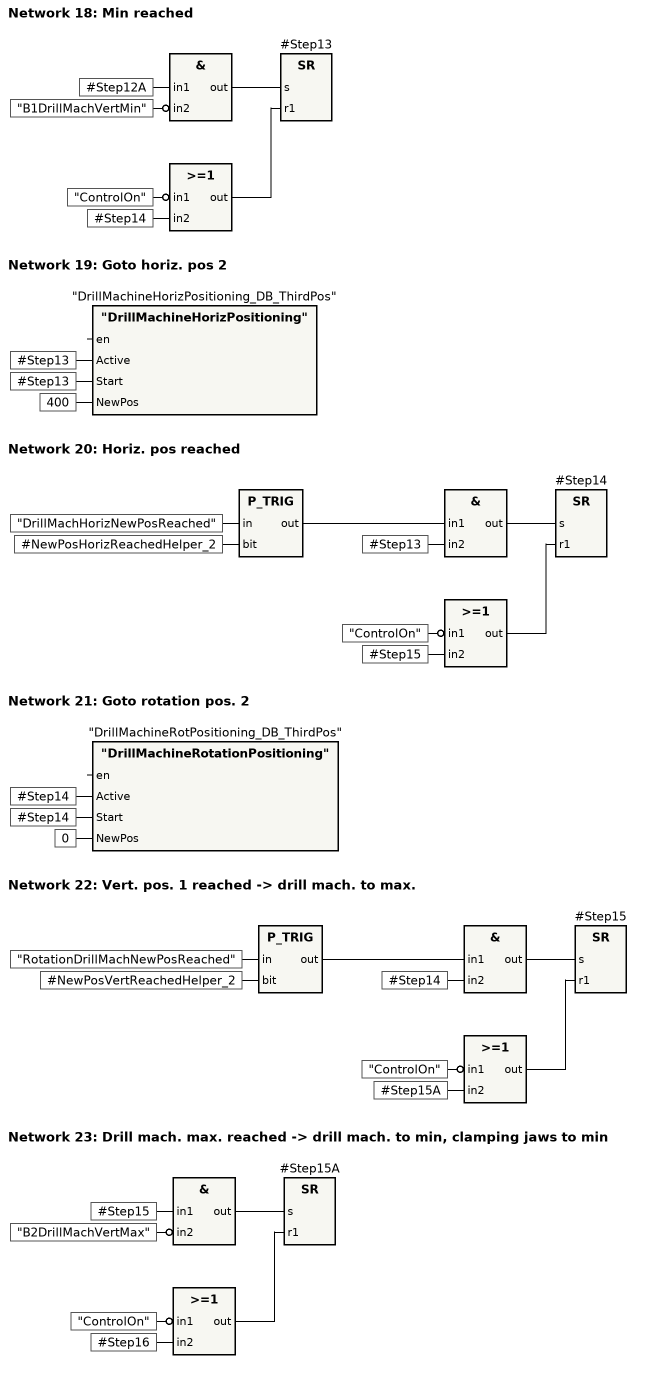
   IF #Step12A AND NOT "B1DrillMachVertMin" THEN
       #Step13 := TRUE;   // SR flip-flop
   END_IF;
   IF NOT "ControlOn" OR #Step14 THEN #Step13 := FALSE; END_IF;
END_REGION

REGION Network 19: Goto horiz. pos 2
   "DrillMachineHorizPositioning_DB_ThirdPos"(Active := #Step13, Start := #Step13, NewPos := 400);   // "DrillMachineHorizPositioning"
END_REGION

REGION Network 20: Horiz. pos reached
   #_w1 := "DrillMachHorizNewPosReached" AND NOT #NewPosHorizReachedHelper_2;   // rising edge
   #NewPosHorizReachedHelper_2 := "DrillMachHorizNewPosReached";
   IF #_w1 AND #Step13 THEN
       #Step14 := TRUE;   // SR flip-flop
   END_IF;
   IF NOT "ControlOn" OR #Step15 THEN #Step14 := FALSE; END_IF;
END_REGION

REGION Network 21: Goto rotation pos. 2
   "DrillMachineRotPositioning_DB_ThirdPos"(Active := #Step14, Start := #Step14, NewPos := 0);   // "DrillMachineRotationPositioning"
END_REGION

REGION Network 22: Vert. pos. 1 reached -> drill mach. to max.
   #_w1 := "RotationDrillMachNewPosReached" AND NOT #NewPosVertReachedHelper_2;   // rising edge
   #NewPosVertReachedHelper_2 := "RotationDrillMachNewPosReached";
   IF #_w1 AND #Step14 THEN
       #Step15 := TRUE;   // SR flip-flop
   END_IF;
   IF NOT "ControlOn" OR #Step15A THEN #Step15 := FALSE; END_IF;
END_REGION

REGION Network 23: Drill mach. max. reached -> drill mach. to min, clamping jaws to min
   IF #Step15 AND NOT "B2DrillMachVertMax" THEN
       #Step15A := TRUE;   // SR flip-flop
   END_IF;
   IF NOT "ControlOn" OR #Step16 THEN #Step15A := FALSE; END_IF;
END_REGION

REGION Network 24: Min reached -> Feed to max.
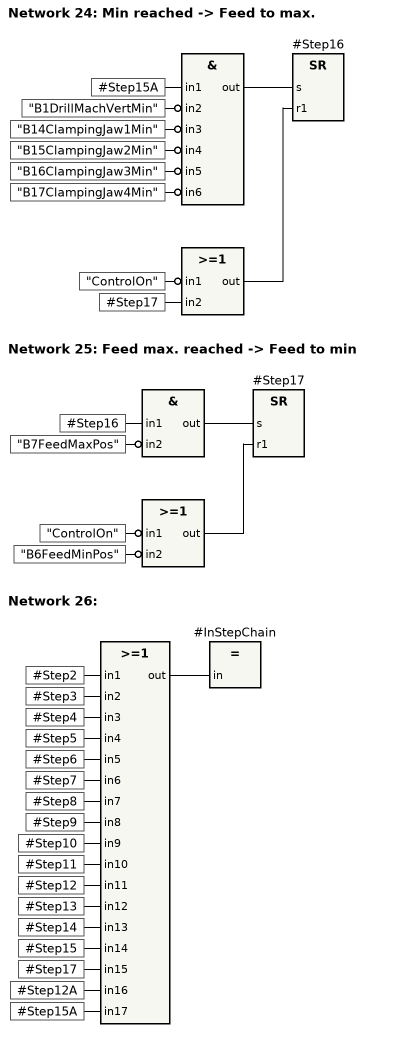
   IF #Step15A AND NOT "B1DrillMachVertMin" AND NOT "B14ClampingJaw1Min" AND NOT "B15ClampingJaw2Min" AND NOT "B16ClampingJaw3Min" AND NOT "B17ClampingJaw4Min" THEN
       #Step16 := TRUE;   // SR flip-flop
   END_IF;
   IF NOT "ControlOn" OR #Step17 THEN #Step16 := FALSE; END_IF;
END_REGION

REGION Network 25: Feed max. reached -> Feed to min
   IF #Step16 AND NOT "B7FeedMaxPos" THEN
       #Step17 := TRUE;   // SR flip-flop
   END_IF;
   IF NOT "ControlOn" OR NOT "B6FeedMinPos" THEN #Step17 := FALSE; END_IF;
END_REGION

REGION Network 26
   #InStepChain := #Step2 OR #Step3 OR #Step4 OR #Step5 OR #Step6 OR #Step7 OR #Step8 OR #Step9 OR #Step10 OR #Step11 OR #Step12 OR #Step13 OR #Step14 OR #Step15 OR #Step17 OR #Step12A OR #Step15A;
END_REGION
END_FUNCTION_BLOCK

FUNCTION_BLOCK "DrillMachineHorizPositioning"   // FB2, FBD
{ S7_Optimized_Access := 'FALSE' }
VERSION : 0.1
   VAR_INPUT
      Active : Bool;
      Start : Bool;
      NewPos : Int := 0;
   END_VAR
   VAR
      PosEdgeStartHelper : Bool;
      PosEdgeStart : Bool;
   END_VAR
   VAR_TEMP   // added for the SCL form of the ladder/FBD networks
      _w1 : Bool;
   END_VAR
BEGIN

REGION Network 1: Active?
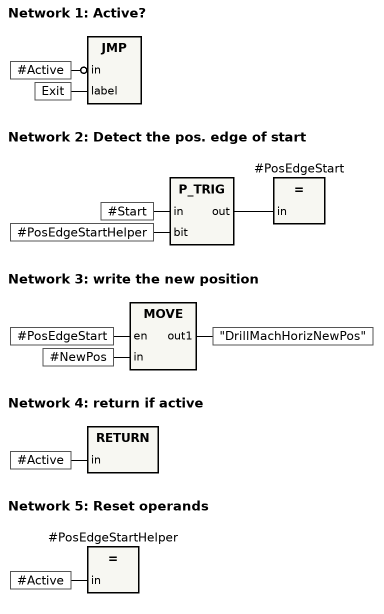
   IF NOT #Active THEN GOTO Exit; END_IF;
END_REGION

REGION Network 2: Detect the pos. edge of start
   #_w1 := #Start AND NOT #PosEdgeStartHelper;   // rising edge
   #PosEdgeStartHelper := #Start;
   #PosEdgeStart := #_w1;
END_REGION

REGION Network 3: write the new position
   IF #PosEdgeStart THEN "DrillMachHorizNewPos" := #NewPos; END_IF;
END_REGION

REGION Network 4: return if active
   IF #Active THEN
       ENO := TRUE;
       RETURN;
   END_IF;
END_REGION

REGION Network 5: Reset operands
   Exit:
   #PosEdgeStartHelper := #Active;
END_REGION
END_FUNCTION_BLOCK

FUNCTION_BLOCK "DrillMachineRotationPositioning"   // FB3, FBD
{ S7_Optimized_Access := 'FALSE' }
VERSION : 0.1
   VAR_INPUT
      Active : Bool;
      Start : Bool;
      NewPos : Int := 0;
   END_VAR
   VAR
      PosEdgeStartHelper : Bool;
      PosEdgeStart : Bool;
   END_VAR
   VAR_TEMP   // added for the SCL form of the ladder/FBD networks
      _w1 : Bool;
   END_VAR
BEGIN

REGION Network 1
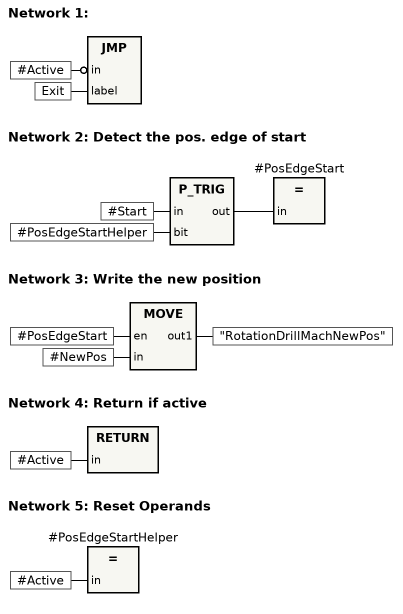
   IF NOT #Active THEN GOTO Exit; END_IF;
END_REGION

REGION Network 2: Detect the pos. edge of start
   #_w1 := #Start AND NOT #PosEdgeStartHelper;   // rising edge
   #PosEdgeStartHelper := #Start;
   #PosEdgeStart := #_w1;
END_REGION

REGION Network 3: Write the new position
   IF #PosEdgeStart THEN "RotationDrillMachNewPos" := #NewPos; END_IF;
END_REGION

REGION Network 4: Return if active
   IF #Active THEN
       ENO := TRUE;
       RETURN;
   END_IF;
END_REGION

REGION Network 5: Reset Operands
   Exit:
   #PosEdgeStartHelper := #Active;
END_REGION
END_FUNCTION_BLOCK

FUNCTION "MHJ-PLC-Lab-Function-S71500" : Void   // FC1, SCL
{ S7_Optimized_Access := 'TRUE' }
VERSION : 0.1
   VAR_INPUT
      MinDiByte : Int;
      MaxDiByte : Int;
   END_VAR
   VAR_TEMP
      Value : Byte;
      ForCounter : Int;
      MaxDiByteTemp : Int;
      MinDiByteTemp : Int;
   END_VAR
   VAR CONSTANT
      Value_01_DW : DWord := 16#1223_5486;
      Value_02_DW : DWord := 16#A6C9_D1F5;
   END_VAR
BEGIN

   #Value:=PEEK(area := 16#82,
        dbNumber := 0,
        byteOffset := 511);
   #Value := #Value + 1;

   POKE(area := 16#82,
        dbNumber := 0,
        byteOffset := 511,
        value := #Value);

   POKE(area := 16#82,
        dbNumber := 0,
        byteOffset := 1016,
        value := #Value_01_DW);
   POKE(area := 16#82,
        dbNumber := 0,
        byteOffset := 1020,
        value := #Value_02_DW);

   #MaxDiByteTemp := 462;
   IF #MaxDiByte < 463 THEN
       #MaxDiByteTemp := #MaxDiByte;
   END_IF;

   #MinDiByteTemp := 0;
   IF #MaxDiByteTemp >= #MinDiByte & #MinDiByte >= 0 THEN
       #MinDiByteTemp := #MinDiByte;
   END_IF;

   FOR #ForCounter := #MinDiByteTemp TO #MaxDiByteTemp DO
       #Value := PEEK(area := 16#1,
                      dbNumber := 0,
                      byteOffset := #ForCounter);
       POKE(area := 16#81,
            dbNumber := 0,
            byteOffset := #ForCounter,
            value := #Value);
   END_FOR;

   #Value := PEEK(area := 16#1,
                  dbNumber := 0,
                  byteOffset := 512);
   POKE(area := 16#82,
        dbNumber := 0,
        byteOffset := 512,
        value := #Value);
END_FUNCTION

FUNCTION "MHJ-PLC-Lab-Function-S71500-NextInputArea" : Void   // FC2, SCL
{ S7_Optimized_Access := 'TRUE' }
VERSION : 0.1
   VAR_INPUT
      MinDiByte : Int;
      MaxDiByte : Int;
   END_VAR
   VAR_TEMP
      Value : Byte;
      ForCounter : Int;
      MaxDiByteTemp : Int;
      MinDiByteTemp : Int;
   END_VAR
BEGIN


   #MaxDiByteTemp := -1;
   IF #MaxDiByte < 463 THEN
       #MaxDiByteTemp := #MaxDiByte;
   END_IF;

   #MinDiByteTemp := -1;
   IF #MaxDiByteTemp >= #MinDiByte & #MinDiByte >= 0 THEN
       #MinDiByteTemp := #MinDiByte;
   END_IF;

   IF #MaxDiByteTemp >= 0 & #MinDiByte >= 0 THEN
       FOR #ForCounter := #MinDiByteTemp TO #MaxDiByteTemp DO
           #Value := PEEK(area := 16#1,
                          dbNumber := 0,
                          byteOffset := #ForCounter);
           POKE(area := 16#81,
                dbNumber := 0,
                byteOffset := #ForCounter,
                value := #Value);
       END_FOR;

   END_IF;
END_FUNCTION

FUNCTION "Settings" : Void   // FC3, FBD
{ S7_Optimized_Access := 'FALSE' }
VERSION : 0.1
BEGIN

REGION Network 1: Slider to max
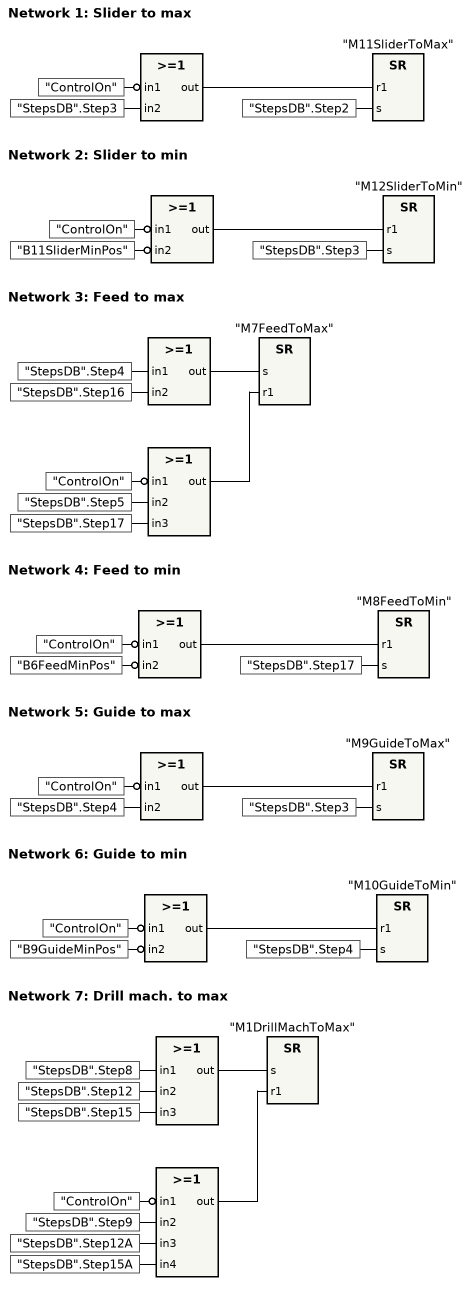
   IF "StepsDB".Step2 THEN
       "M11SliderToMax" := TRUE;   // SR flip-flop
   END_IF;
   IF NOT "ControlOn" OR "StepsDB".Step3 THEN "M11SliderToMax" := FALSE; END_IF;
END_REGION

REGION Network 2: Slider to min
   IF "StepsDB".Step3 THEN
       "M12SliderToMin" := TRUE;   // SR flip-flop
   END_IF;
   IF NOT "ControlOn" OR NOT "B11SliderMinPos" THEN "M12SliderToMin" := FALSE; END_IF;
END_REGION

REGION Network 3: Feed to max
   IF "StepsDB".Step4 OR "StepsDB".Step16 THEN
       "M7FeedToMax" := TRUE;   // SR flip-flop
   END_IF;
   IF NOT "ControlOn" OR "StepsDB".Step5 OR "StepsDB".Step17 THEN "M7FeedToMax" := FALSE; END_IF;
END_REGION

REGION Network 4: Feed to min
   IF "StepsDB".Step17 THEN
       "M8FeedToMin" := TRUE;   // SR flip-flop
   END_IF;
   IF NOT "ControlOn" OR NOT "B6FeedMinPos" THEN "M8FeedToMin" := FALSE; END_IF;
END_REGION

REGION Network 5: Guide to max
   IF "StepsDB".Step3 THEN
       "M9GuideToMax" := TRUE;   // SR flip-flop
   END_IF;
   IF NOT "ControlOn" OR "StepsDB".Step4 THEN "M9GuideToMax" := FALSE; END_IF;
END_REGION

REGION Network 6: Guide to min
   IF "StepsDB".Step4 THEN
       "M10GuideToMin" := TRUE;   // SR flip-flop
   END_IF;
   IF NOT "ControlOn" OR NOT "B9GuideMinPos" THEN "M10GuideToMin" := FALSE; END_IF;
END_REGION

REGION Network 7: Drill mach. to max
   IF "StepsDB".Step8 OR "StepsDB".Step12 OR "StepsDB".Step15 THEN
       "M1DrillMachToMax" := TRUE;   // SR flip-flop
   END_IF;
   IF NOT "ControlOn" OR "StepsDB".Step9 OR "StepsDB".Step12A OR "StepsDB".Step15A THEN
       "M1DrillMachToMax" := FALSE;
   END_IF;
END_REGION

REGION Network 8: Drill mach. to min
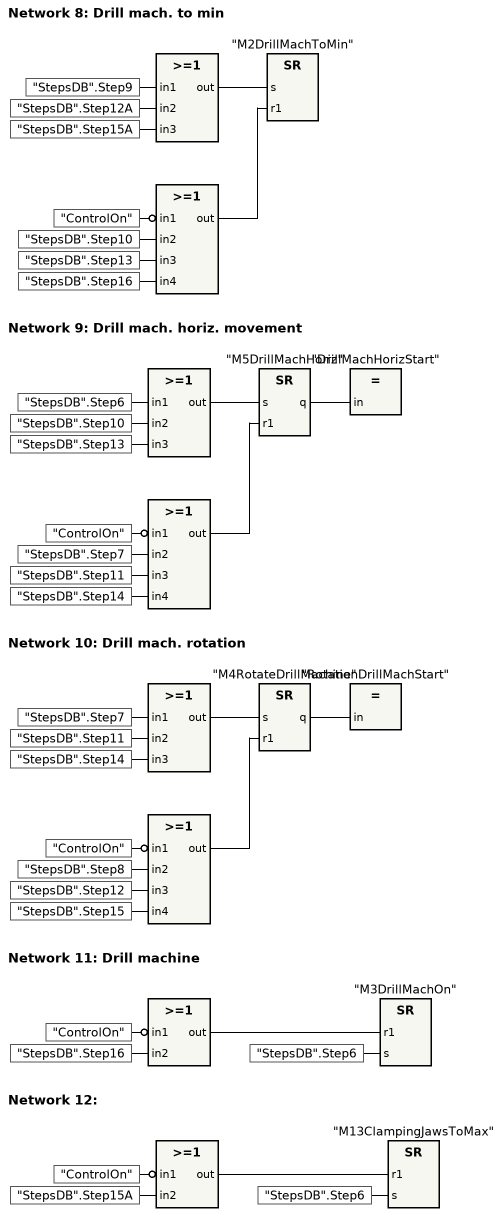
   IF "StepsDB".Step9 OR "StepsDB".Step12A OR "StepsDB".Step15A THEN
       "M2DrillMachToMin" := TRUE;   // SR flip-flop
   END_IF;
   IF NOT "ControlOn" OR "StepsDB".Step10 OR "StepsDB".Step13 OR "StepsDB".Step16 THEN
       "M2DrillMachToMin" := FALSE;
   END_IF;
END_REGION

REGION Network 9: Drill mach. horiz. movement
   IF "StepsDB".Step6 OR "StepsDB".Step10 OR "StepsDB".Step13 THEN
       "M5DrillMachHoriz" := TRUE;   // SR flip-flop
   END_IF;
   IF NOT "ControlOn" OR "StepsDB".Step7 OR "StepsDB".Step11 OR "StepsDB".Step14 THEN
       "M5DrillMachHoriz" := FALSE;
   END_IF;
   "DrillMachHorizStart" := "M5DrillMachHoriz";
END_REGION

REGION Network 10: Drill mach. rotation
   IF "StepsDB".Step7 OR "StepsDB".Step11 OR "StepsDB".Step14 THEN
       "M4RotateDrillMachine" := TRUE;   // SR flip-flop
   END_IF;
   IF NOT "ControlOn" OR "StepsDB".Step8 OR "StepsDB".Step12 OR "StepsDB".Step15 THEN
       "M4RotateDrillMachine" := FALSE;
   END_IF;
   "RotationDrillMachStart" := "M4RotateDrillMachine";
END_REGION

REGION Network 11: Drill machine
   IF "StepsDB".Step6 THEN
       "M3DrillMachOn" := TRUE;   // SR flip-flop
   END_IF;
   IF NOT "ControlOn" OR "StepsDB".Step16 THEN "M3DrillMachOn" := FALSE; END_IF;
END_REGION

REGION Network 12
   IF "StepsDB".Step6 THEN
       "M13ClampingJawsToMax" := TRUE;   // SR flip-flop
   END_IF;
   IF NOT "ControlOn" OR "StepsDB".Step15A THEN "M13ClampingJawsToMax" := FALSE; END_IF;
END_REGION
END_FUNCTION

ORGANIZATION_BLOCK "Main"   // OB1, FBD, ProgramCycle
TITLE = "Main Program Sweep (Cycle)"
{ S7_Optimized_Access := 'FALSE' }
VERSION : 0.1
   VAR_TEMP
      OB1_EV_CLASS : Byte;   // Bits 0-3 = 1 (Coming event), Bits 4-7 = 1 (Event class 1)
      OB1_SCAN_1 : Byte;   // 1 (Cold restart scan 1 of OB 1), 3 (Scan 2-n of OB 1)
      OB1_PRIORITY : Byte;   // Priority of OB Execution
      OB1_OB_NUMBR : Byte;   // 1 (Organization block 1, OB1)
      OB1_RESERVED_1 : Byte;   // Reserved for system
      OB1_RESERVED_2 : Byte;   // Reserved for system
      OB1_PREV_CYCLE : Int;   // Cycle time of previous OB1 scan (milliseconds)
      OB1_MIN_CYCLE : Int;   // Minimum cycle time of OB1 (milliseconds)
      OB1_MAX_CYCLE : Int;   // Maximum cycle time of OB1 (milliseconds)
      OB1_DATE_TIME : Date_And_Time;   // Date and time OB1 started
   END_VAR
   VAR_TEMP   // added for the SCL form of the ladder/FBD networks
      _w1 : Bool;
   END_VAR
BEGIN

REGION Network 1
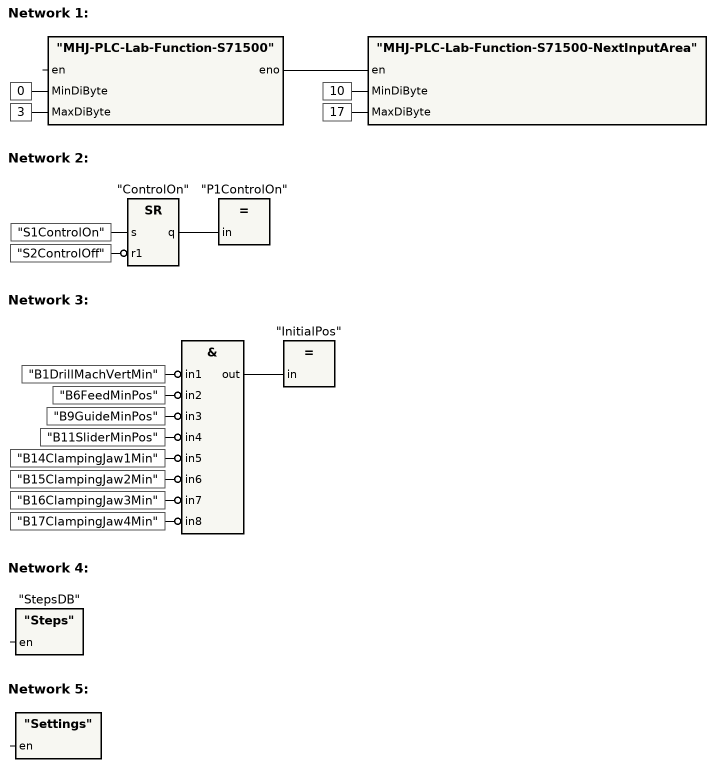
   "MHJ-PLC-Lab-Function-S71500"(MinDiByte := 0, MaxDiByte := 3, ENO => #_w1);
   IF #_w1 THEN "MHJ-PLC-Lab-Function-S71500-NextInputArea"(MinDiByte := 10, MaxDiByte := 17); END_IF;
END_REGION

REGION Network 2
   IF "S1ControlOn" THEN
       "ControlOn" := TRUE;   // SR flip-flop
   END_IF;
   IF NOT "S2ControlOff" THEN "ControlOn" := FALSE; END_IF;
   "P1ControlOn" := "ControlOn";
END_REGION

REGION Network 3
   "InitialPos" := NOT "B1DrillMachVertMin" AND NOT "B6FeedMinPos" AND NOT "B9GuideMinPos" AND NOT "B11SliderMinPos" AND NOT "B14ClampingJaw1Min" AND NOT "B15ClampingJaw2Min" AND NOT "B16ClampingJaw3Min" AND NOT "B17ClampingJaw4Min";
END_REGION

REGION Network 4
   "StepsDB"();   // "Steps"
END_REGION

REGION Network 5
   "Settings"();
END_REGION
END_ORGANIZATION_BLOCK